TYPE RfidConfigs :
STRUCT
	BisL405RfidConfig : BisL405RfidConfig;
END_STRUCT
END_TYPE

(* stored: Version 1.1.0.1, ProductVersion 3.1.4024.12
   DUT RfidConfigs: Id {ab437621-ef37-49fb-adcf-6509d35c0805} *)
